(* CoDeSys 2.3 export: ROBOT_STATE.EXP *)

(* Data type in Robot *)
TYPE ROBOT_STATE :
STRUCT
	Enabled : BOOL;
	Simulation : BOOL;
	Ready : BOOL;
	Busy : BOOL;
	Error : BOOL;
	Ack : BOOL;
	PickDone : BOOL;
	PickFailed : BOOL;
	CurrentTargetId : INT;
	ErrorCode : UINT;
END_STRUCT
END_TYPE
